// TIA Portal V20 export
TYPE "typeFDoorElement"
// stored: Access Published, IsFailsafeCompliant true, Namespace Safety
   STRUCT
      FDoor1 : Bool;
      FDoor2 : Bool;
      FDoor3 : Bool;
      FDoor4 : Bool;
      FDoor5 : Bool;
      FDoor6 : Bool;
      FDoor7 : Bool;
      FDoor8 : Bool;
      FDoor9 : Bool;
      FDoor10 : Bool;
   END_STRUCT;
END_TYPE
